INTERFACE I_HE_SATT_FilterHolder


METHOD GetFilter : I_HE_SATT_Filter
VAR_INPUT
    nFilterNumber : INT;
END_VAR
END_METHOD


METHOD MoveToFilter
VAR_INPUT
    iFilter : I_HE_SATT_Filter;
    fThickness : LREAL;
END_VAR
END_METHOD


PROPERTY NumberOfSlots : INT
GET
END_GET
END_PROPERTY


METHOD RegisterFilter
VAR_INPUT
    iFilter : I_HE_SATT_Filter;
END_VAR
END_METHOD


PROPERTY Status : REFERENCE TO ST_HE_SATT_Status
GET
END_GET
END_PROPERTY

END_INTERFACE

(* stored: Version 1.1.0.1
   Itf I_HE_SATT_FilterHolder: Id {50894da0-cc33-47a4-8023-07412f59bfc3}
   Method GetFilter: Id {b9af26ac-850d-4c8d-8479-197f9f19bd28}
   Method MoveToFilter: Id {42d2d649-ec14-4b4d-9b6b-ac71b890eebc}
   Property NumberOfSlots: Id {e83b7fb5-7407-4813-b9cc-d270aebd7af9}
   Get Get: Id {3b73d66b-ce03-4755-bc84-99831ecd961a}
   Method RegisterFilter: Id {120292f7-d437-453b-8f04-99e161e38474}
   Property Status: Id {838e8368-38e8-4eb9-851f-0c929494f5e3}
   Get Get: Id {39407399-1ad2-4709-8508-ecccc47d1e58} *)
